Staubli VAL3: InitSysIO.pgx

public program InitSysIO()
// Inialize system io's
begin
  //\private
  call SysIN()
  call SysOUT()
end
